FUNCTION_BLOCK FB_VFD_Mdriver EXTENDS FB_UniversalVFDModbus

VAR
	eFaultInfor	: E_VfdMdriverFaultInfor;
END_VAR

//bError := eVfdStatus
SUPER^();

METHOD Convert : BOOL
VAR_INPUT
	iRegionNo	:	INT;
	pReadData	:	POINTER TO word;
END_VAR
CASE	iRegionNo OF
	0: 
	
		lrHzActual		:= WORD_TO_LREAL( pReadData[0])*0.01;	//4097	/unit /100
		lrDcVoltage		:= WORD_TO_LREAL( pReadData[1])*0.1;	//4098 	/10
		lrVacOutToMotor	:= WORD_TO_LREAL( pReadData[2]);	//4099	/1
		lrCurrent		:= WORD_TO_LREAL(  pReadData[3])*0.01;		//4100	/100
		//4 reserve
		lrPowerKw		:= WORD_TO_LREAL(  pReadData[5])*0.001;		//4102	/1000> kW
	
	1: // status
		CASE pReadData[0] OF
			0: eVfdStatus := VFD_STATUS_STOP;
			
			1: 
				eVfdStatus := VFD_STATUS_RUNNING_FORWARD;
			2:
				eVfdStatus := VFD_STATUS_RUNNING_REVERSE;
			3: 
				eVfdStatus := VFD_STATUS_STOP;
		END_CASE
		// important
		IF eVfdState = VFD_INITIALIZING THEN
			IF eFaultInfor = E_VfdMdriverFaultInfor.Nofault
			AND eVfdStatus = VFD_STATUS_STOP THEN
				eVfdStatus := VFD_STATUS_READY_TO_RUN;
			ELSIF eFaultInfor <> E_VfdMdriverFaultInfor.Nofault THEN
				eVfdStatus := VFD_STATUS_FAULT;
			END_IF
		END_IF
		IF eFaultInfor <> E_VfdMdriverFaultInfor.Nofault THEN
			eVfdStatus := VFD_STATUS_FAULT;
		END_IF
		IF iModbusErrorID = MODBUSERROR_C_NO_RESPONSE THEN
			eVfdStatus := VFD_STATUS_NOT_RESPOND;
		END_IF
		// important
	
	2: 
	
		iErrorID := WORD_TO_UDINT( pReadData[0]);
		eFaultInfor :=  WORD_TO_UINT( pReadData[0]);
END_CASE
END_METHOD

METHOD  FirstCycle 
VAR_INPUT
	sName : STRING;
	iUnitID : BYTE ; // modbus address of the device : 1- 255
END_VAR
SUPER^.FirstCycle( sName := sName, iUnitID := iUnitID);
(*Assign Ctrol Word : user Manual M-driver*)
VFD_CTRL_RESET_FAULT := 7;
VFD_CTRL_RUN_FORWARD := 1;
VFD_CTRL_RUN_REVERSE := 2;
VFD_CTRL_STOP_FREE 		:= 5;
VFD_CTRL_STOP_SPEED_DOWN	:= 6;
///  actual hz, current, voltage
arrAddressRead[0][0] := 4097;
arrAddressRead[0][1]	:= 6;
arrAddressRead[0][2]	:= E_ModbusFunction.ReadHoldingRegisters;

// actual state	
arrAddressRead[1][0] := 16#3000;
arrAddressRead[1][1]	:= 1;
arrAddressRead[1][2]	:= E_ModbusFunction.ReadHoldingRegisters;

// fault infor
arrAddressRead[2][0] := 16#8000;
arrAddressRead[2][1]	:= 1;
arrAddressRead[2][2]	:= E_ModbusFunction.ReadHoldingRegisters;

iNumAddRegionRead	:= 3;

/////write control WORD VFD
arrAddressWrite[iCTRL_WORD][0]	:= 16#2000;
arrAddressWrite[iCTRL_WORD][1]	:= 1;
arrAddressWrite[iCTRL_WORD][2]	:= VFD_CTRL_STOP_FREE;
arrAddressWrite[iCTRL_WORD][10]	:= E_ModbusFunction.WriteSingleRegister;
// Frequency
arrAddressWrite[iCTRL_FREQUENCY_WORD][0]	:= 4096;
arrAddressWrite[iCTRL_FREQUENCY_WORD][1]	:= 1;
							(*MUST BE CARE FULL WHEN USE FLOATING POINT CONVERT*)
arrAddressWrite[iCTRL_FREQUENCY_WORD][2]	:= LREAL_TO_WORD( F_ScaleValue(	rangeRawMin := 0,
															rangeRawMax := 50,
															RangeScaleMin :=0,
															RangeScaleMax := 10000,
															ValueRaw := 0)
										  );
arrAddressWrite[iCTRL_FREQUENCY_WORD][10]	:= E_ModbusFunction.WriteSingleRegister;
										  
iNumAddRegionWrite := 2;
END_METHOD

METHOD PROTECTED  MS_Aborting
arrAddressWrite[iCTRL_WORD][2]	:= VFD_CTRL_STOP_FREE;
SUPER^.MS_Aborting();
END_METHOD

METHOD PROTECTED  MS_RunForward
VAR_INPUT
END_VAR
arrAddressWrite[iCTRL_FREQUENCY_WORD][2] :=  LREAL_TO_WORD( 
															F_ScaleValue(	rangeRawMin := 0,
																			rangeRawMax := 50,
																			RangeScaleMin := 0,
																			RangeScaleMax := 10000,
																			ValueRaw := lrHzControl) 
																				);
SUPER^.MS_RunForward();
END_METHOD

METHOD PROTECTED  MS_RunReverse
VAR_INPUT
END_VAR
arrAddressWrite[iCTRL_FREQUENCY_WORD][2] :=  LREAL_TO_WORD( 
															F_ScaleValue(	rangeRawMin := 0,
																			rangeRawMax := 50,
																			RangeScaleMin := 0,
																			RangeScaleMax := 10000,
																			ValueRaw := lrHzControl) 
																				);
SUPER^.MS_RunReverse();
END_METHOD

END_FUNCTION_BLOCK

(* stored: Version 1.1.0.1, ProductVersion 3.1.4024.12
   POU FB_VFD_Mdriver: Id {a6c61530-0033-4638-a4bf-9e8688f84f90}, SpecialFunc None
   Method Convert: Id {fafa2ce9-b6ea-4be6-a0f9-88bd4e57300b}
   Method FirstCycle: Id {6a7a0af9-8902-465d-a9dd-89f6088e46db}
   Method MS_Aborting: Id {3105377d-b85b-4bca-a7cf-3ef8c0a5e8bb}
   Method MS_RunForward: Id {628dc59e-846e-40d0-9cf1-88b6513e9da9}
   Method MS_RunReverse: Id {f2f7d6df-b61b-4d5f-95b3-bdaa7e913b8f} *)
